(* IEC 61131-3 sources: ST/Codesys_ZWB, 2 files *)

(* ---- calclRezhim1.st ---- *)
PROGRAM calclRezhim1

VAR_INPUT
    konf_SA_Pusk_Stop : BOOL;
    P_rezhim_ypr : INT;
    Alarm_critical : BOOL;
    Di_sa_pusk_stop : BOOL;

    otM_Pusk : BOOL;
    otM_Stop : BOOL;
END_VAR

VAR_OUTPUT
    rezhim1 : BOOL;
END_VAR

// вычисление режима установки
IF konf_SA_Pusk_Stop = FALSE THEN
    P_rezhim_ypr := 1;
    // если переключателя пуск/стоп не предусмотрено, то переходим в режим управления дистанционный
    // и ждём команды на запуск от мастера
END_IF;

IF P_rezhim_ypr = 0 AND konf_SA_Pusk_Stop = TRUE THEN
    // если режим управления местный и есть переключатель пуск/стоп
    IF Alarm_critical = TRUE OR Di_sa_pusk_stop = FALSE THEN
        rezhim1 := FALSE;
    END_IF;
    IF Alarm_critical <> TRUE AND Di_sa_pusk_stop = TRUE THEN
        rezhim1 := TRUE;
    END_IF;
END_IF;

IF P_rezhim_ypr = 1 AND konf_SA_Pusk_Stop = TRUE THEN
    // режим дистанционный и есть переключатель пуск/стоп
    IF Di_sa_pusk_stop = TRUE THEN
        IF Alarm_critical = TRUE THEN
            rezhim1 := FALSE;
        END_IF;
        IF Alarm_critical <> TRUE AND otM_Pusk = TRUE THEN
            rezhim1 := TRUE;
            otM_Pusk := FALSE;
        END_IF;
        IF Alarm_critical <> TRUE AND otM_Stop = TRUE THEN
            rezhim1 := FALSE;
            otM_Stop := FALSE;
        END_IF;
    END_IF;
    IF Di_sa_pusk_stop = FALSE THEN
        rezhim1 := FALSE;
    END_IF;
END_IF;

IF P_rezhim_ypr = 1 AND konf_SA_Pusk_Stop = FALSE THEN
    // режим дистанционный и нет переключателя пуск/стоп
    IF Alarm_critical = TRUE THEN
        rezhim1 := FALSE;
    END_IF;
    IF Alarm_critical <> TRUE AND otM_Pusk = TRUE THEN
        rezhim1 := TRUE;
        otM_Pusk := FALSE;
    END_IF;
    IF Alarm_critical <> TRUE AND otM_Stop = TRUE THEN
        rezhim1 := FALSE;
        otM_Stop := FALSE;
    END_IF;
END_IF;
END_PROGRAM

(* ---- VoKal_v1r1.st ---- *)
PROGRAM VoKal

VAR_INPUT
    Komanda: INT;
    vremya_goda: INT;
    Tobr: REAL;
    N_Tobr_prog_let: REAL;
    N_Tobr_prog_zim: REAL;
    init_end: BOOL;
    rezhim1: INT;
    rezhim2: INT;
    Di_QF_Nasos: BOOL;
    Di_TS_VoKal: BOOL;
    N_niz_Tobr_let: REAL;
    N_niz_Tobr_zim: REAL;
END_VAR

VAR_OUTPUT
    Do_Nasos: BOOL;
    VK_progret: BOOL;
    A_net_pitaniya_Nasos: BOOL;
    A_Ygroza_zamorozki_TS: BOOL;
    A_Ygroza_zamorozki_Tpr: BOOL;
    A_Ygroza_zamorozki_Tobr: BOOL;
    A_Ygroza_zamorozki: BOOL;
END_VAR

VAR
    Init: INT := 0; // Инициализация
    Dezh: INT := 1; // Дежурный
    Preheat: INT := 2; // Предпрогрев
    Run: INT := 3; // Работа
    Prodyv: INT := 4; // Продувка
    Alarm: INT := 5; // Авария
    Block: INT := 6; // Блокировка
    Enable: BOOL; // Разрешение
END_VAR

IF vremya_goda = 0 AND Tobr > N_Tobr_prog_let AND init_end = TRUE AND rezhim2 = Preheat THEN
    VK_progret := TRUE;
END_IF;

IF vremya_goda = 1 AND Tobr > N_Tobr_prog_zim AND init_end = TRUE AND rezhim2 = Preheat THEN
    VK_progret := TRUE;
END_IF;

IF rezhim1 = 0 THEN (* Режим1 останов *)
    VK_progret := FALSE;
END_IF;

IF vremya_goda = 1 AND Di_QF_Nasos = TRUE THEN
    (* доделать *)
    Do_Nasos := TRUE;
END_IF;

IF vremya_goda = 0 THEN
    (* доделать *)
    Do_Nasos := FALSE;
END_IF;

IF Di_QF_Nasos = FALSE AND init_end = TRUE THEN
    (* доделать *)
    Do_Nasos := FALSE;
    A_net_pitaniya_Nasos := TRUE;
ELSE
    A_net_pitaniya_Nasos := FALSE;
END_IF;

IF Di_TS_VoKal = FALSE AND init_end = TRUE THEN
    A_Ygroza_zamorozki_TS := TRUE;
END_IF;

IF Di_TS_VoKal = TRUE AND init_end = TRUE THEN
    (* && Reset_alarm = TRUE *)
    A_Ygroza_zamorozki_TS := FALSE;
END_IF;

IF A_Ygroza_zamorozki_TS = TRUE OR A_Ygroza_zamorozki_Tpr = TRUE OR A_Ygroza_zamorozki_Tobr = TRUE THEN
    A_Ygroza_zamorozki := TRUE;
ELSE
    A_Ygroza_zamorozki := FALSE;
END_IF;

IF vremya_goda = 0 AND init_end = TRUE AND Tobr < N_niz_Tobr_let THEN
    A_Ygroza_zamorozki_Tobr := TRUE;
END_IF;

IF vremya_goda = 1 AND init_end = TRUE AND Tobr < N_niz_Tobr_zim THEN
    A_Ygroza_zamorozki_Tobr := TRUE;
END_IF;

IF vremya_goda = 0 AND init_end = TRUE AND Tobr >= N_Tobr_prog_let THEN
    A_Ygroza_zamorozki_Tobr := FALSE;
END_IF;

IF vremya_goda = 1 AND init_end = TRUE AND Tobr >= N_Tobr_prog_zim THEN
    A_Ygroza_zamorozki_Tobr := FALSE;
END_IF;

IF N_niz_Tobr_let + 5 > N_Tobr_prog_let THEN
    N_Tobr_prog_let := N_niz_Tobr_let + 5;
END_IF;

IF N_niz_Tobr_zim + 5 > N_Tobr_prog_zim THEN
    N_Tobr_prog_zim := N_niz_Tobr_zim + 5;
END_IF;

END_PROGRAM
